(* IEC 61131-3 sources: volt/packages/volt-lsp-iec/test-corpus/pro2193/Device/Plc Logic/Application/09 Misc/Library Manager/SysTask, 36 files *)

(* ---- PFSYS_TASK_EXCEPTIONHANDLER.dut ---- *)
TYPE PFSYS_TASK_EXCEPTIONHANDLER : POINTER TO BYTE;
END_TYPE

(* ---- PFSYS_TASK_FUNCTION.dut ---- *)
TYPE PFSYS_TASK_FUNCTION : POINTER TO BYTE;
END_TYPE

(* ---- REGCONTEXT.dut ---- *)
TYPE REGCONTEXT :
STRUCT
	ULIP : __UXINT;
	ULBP : __UXINT;
	ULSP : __UXINT;
END_STRUCT
END_TYPE

(* ---- SYS_TASK_INFO.dut ---- *)
TYPE SYS_TASK_INFO :
STRUCT
	UIOSHANDLE : RTS_IEC_HANDLE;
	ISTATE : DINT;
	IOLDSTATE : DINT;
	TP : SYS_TASK_PARAM;
	ULCYCLETIME : UDINT;
	ULCYCLESTART : UDINT;
	ULPRIORITY : UDINT;
	ULOSPRIORITY : UDINT;
	ULINTERVAL : UDINT;
	ULSTACKSIZE : UDINT;
	PFUNCTION : PFSYS_TASK_FUNCTION;
	SZNAME : STRING(SYSTASK_MAX_NAME_LEN);
	PEXCEPTIONHANDLER : PFSYS_TASK_EXCEPTIONHANDLER;
	CONTEXT : RegContext;
	PCPPINSTANCE : POINTER TO BYTE;
	POSSPECIFIC : POINTER TO BYTE;
	ULFEATURE : DWORD;
END_STRUCT
END_TYPE

(* ---- SYS_TASK_PARAM.dut ---- *)
TYPE SYS_TASK_PARAM :
STRUCT
	HTASK : RTS_IEC_HANDLE;
	BEXIT : DINT;
	ULINTERVAL : UDINT;
	PPARAM : POINTER TO BYTE;
END_STRUCT
END_TYPE

(* ---- FEATUREFLAGS.gvl ---- *)
VAR_GLOBAL
	SYSTASK_FF_NONE : DWORD := 16#0;
	SYSTASK_FF_AUTORELEASEONEXIT : DWORD := 16#1;
END_VAR

(* ---- GVL.gvl ---- *)
VAR_GLOBAL
	SYSTASK_MAX_NAME_LEN : UDINT := 19;
END_VAR

(* ---- TASKPRIORITIES.gvl ---- *)
VAR_GLOBAL
	TASKPRIO_RANGE : UDINT := 255;
	TASKPRIO_SEGMENT : UDINT := 32;
	TASKPRIO_MAX : UDINT := 0;
	TASKPRIO_SYSTEM_BASE : UDINT := 0;
	TASKPRIO_SYSTEM_END : UDINT := 31;
	TASKPRIO_REALTIME_BASE : UDINT := 32;
	TASKPRIO_REALTIME_END : UDINT := 63;
	TASKPRIO_HIGH_BASE : UDINT := 64;
	TASKPRIO_HIGH_END : UDINT := 95;
	TASKPRIO_ABOVENORMAL_BASE : UDINT := 96;
	TASKPRIO_ABOVENORMAL_END : UDINT := 127;
	TASKPRIO_NORMAL_BASE : UDINT := 128;
	TASKPRIO_NORMAL_END : UDINT := 159;
	TASKPRIO_BELOWNORMAL_BASE : UDINT := 160;
	TASKPRIO_BELOWNORMAL_END : UDINT := 191;
	TASKPRIO_LOW_BASE : UDINT := 192;
	TASKPRIO_LOW_END : UDINT := 223;
	TASKPRIO_LOWEST_BASE : UDINT := 224;
	TASKPRIO_LOWEST_END : UDINT := 255;
	TASKPRIO_IDLE : UDINT := 255;
	TASKPRIO_MIN : UDINT := 255;
END_VAR

(* ---- SYSTASKAUTORELEASEONEXIT.pou ---- *)
FUNCTION SYSTASKAUTORELEASEONEXIT : RTS_IEC_RESULT
VAR_INPUT
	HTASK : RTS_IEC_HANDLE;
END_VAR
END_FUNCTION

(* ---- SYSTASKCHECKSTACK.pou ---- *)
FUNCTION SYSTASKCHECKSTACK : RTS_IEC_RESULT
VAR_INPUT
	HTASK : RTS_IEC_HANDLE;
	PULMAXDEPTH : POINTER TO UDINT;
END_VAR
END_FUNCTION

(* ---- SYSTASKCREATE.pou ---- *)
FUNCTION SYSTASKCREATE : RTS_IEC_RESULT
VAR_INPUT
	PSZTASKNAME : REFERENCE TO STRING;
	PFUNCTION : PFSYS_TASK_FUNCTION;
	PPARAM : POINTER TO SYS_TASK_PARAM;
	ULPRIORITY : UDINT;
	ULINTERVAL : UDINT;
	ULSTACKSIZE : UDINT;
	PEXCEPTIONHANDLER : PFSYS_TASK_EXCEPTIONHANDLER;
	PHTASKHANDLE : POINTER TO RTS_IEC_HANDLE;
END_VAR
END_FUNCTION

(* ---- SYSTASKCREATE2.pou ---- *)
FUNCTION SYSTASKCREATE2 : RTS_IEC_HANDLE
VAR_INPUT
	PSZTASKNAME : REFERENCE TO STRING;
	PFUNCTION : PFSYS_TASK_FUNCTION;
	PPARAM : POINTER TO SYS_TASK_PARAM;
	ULPRIORITY : UDINT;
	ULINTERVAL : UDINT;
	ULSTACKSIZE : UDINT;
	PEXCEPTIONHANDLER : PFSYS_TASK_EXCEPTIONHANDLER;
	PRESULT : POINTER TO RTS_IEC_RESULT;
END_VAR
END_FUNCTION

(* ---- SYSTASKDESTROY.pou ---- *)
FUNCTION SYSTASKDESTROY : RTS_IEC_RESULT
VAR_INPUT
	HTASK : RTS_IEC_HANDLE;
END_VAR
END_FUNCTION

(* ---- SYSTASKEND.pou ---- *)
FUNCTION SYSTASKEND : RTS_IEC_RESULT
VAR_INPUT
	HTASK : RTS_IEC_HANDLE;
	ULEXITCODE : UDINT;
END_VAR
END_FUNCTION

(* ---- SYSTASKENTER.pou ---- *)
FUNCTION SYSTASKENTER : RTS_IEC_RESULT
VAR_INPUT
	HTASK : RTS_IEC_HANDLE;
END_VAR
END_FUNCTION

(* ---- SYSTASKEXIT.pou ---- *)
FUNCTION SYSTASKEXIT : RTS_IEC_RESULT
VAR_INPUT
	HTASK : RTS_IEC_HANDLE;
	ULTIMEOUTMS : UDINT;
END_VAR
END_FUNCTION

(* ---- SYSTASKGENERATEEXCEPTION.pou ---- *)
FUNCTION SYSTASKGENERATEEXCEPTION : RTS_IEC_RESULT
VAR_INPUT
	ULTASKOSHANDLE : RTS_IEC_HANDLE;
	ULEXCEPTION : UDINT;
	CONTEXT : RegContext;
END_VAR
END_FUNCTION

(* ---- SYSTASKGETCONTEXT.pou ---- *)
FUNCTION SYSTASKGETCONTEXT : RTS_IEC_RESULT
VAR_INPUT
	HTASK : RTS_IEC_HANDLE;
	PCONTEXT : POINTER TO RegContext;
END_VAR
END_FUNCTION

(* ---- SYSTASKGETCURRENT.pou ---- *)
FUNCTION SYSTASKGETCURRENT : RTS_IEC_RESULT
VAR_INPUT
	PHTASK : POINTER TO RTS_IEC_HANDLE;
END_VAR
END_FUNCTION

(* ---- SYSTASKGETCURRENTOSHANDLE.pou ---- *)
FUNCTION SYSTASKGETCURRENTOSHANDLE : RTS_IEC_RESULT
VAR_INPUT
	PUITASKOSHANDLE : POINTER TO RTS_IEC_HANDLE;
END_VAR
END_FUNCTION

(* ---- SYSTASKGETINFO.pou ---- *)
FUNCTION SYSTASKGETINFO : RTS_IEC_RESULT
VAR_INPUT
	HTASK : RTS_IEC_HANDLE;
	PPINFO : POINTER TO POINTER TO SYS_TASK_INFO;
END_VAR
END_FUNCTION

(* ---- SYSTASKGETINTERVAL.pou ---- *)
FUNCTION SYSTASKGETINTERVAL : RTS_IEC_RESULT
VAR_INPUT
	HTASK : RTS_IEC_HANDLE;
END_VAR
VAR_IN_OUT
	PULINTERVAL : UDINT;
END_VAR
END_FUNCTION

(* ---- SYSTASKGETNAME.pou ---- *)
FUNCTION SYSTASKGETNAME : POINTER TO STRING
VAR_INPUT
	HTASK : RTS_IEC_HANDLE;
	PRESULT : POINTER TO RTS_IEC_RESULT;
END_VAR
END_FUNCTION

(* ---- SYSTASKGETOSHANDLE.pou ---- *)
FUNCTION SYSTASKGETOSHANDLE : RTS_IEC_HANDLE
VAR_INPUT
	HTASK : RTS_IEC_HANDLE;
END_VAR
END_FUNCTION

(* ---- SYSTASKGETOSPRIORITY.pou ---- *)
FUNCTION SYSTASKGETOSPRIORITY : RTS_IEC_RESULT
VAR_INPUT
	HTASK : RTS_IEC_HANDLE;
	PULOSPRIORITY : POINTER TO UDINT;
END_VAR
END_FUNCTION

(* ---- SYSTASKGETPRIORITY.pou ---- *)
FUNCTION SYSTASKGETPRIORITY : RTS_IEC_RESULT
VAR_INPUT
	HTASK : RTS_IEC_HANDLE;
	PULPRIORITY : POINTER TO UDINT;
END_VAR
END_FUNCTION

(* ---- SYSTASKJOIN.pou ---- *)
FUNCTION SYSTASKJOIN : RTS_IEC_RESULT
VAR_INPUT
	HTASKTOJOIN : RTS_IEC_HANDLE;
	ULTIMEOUTMS : UDINT;
END_VAR
END_FUNCTION

(* ---- SYSTASKLEAVE.pou ---- *)
FUNCTION SYSTASKLEAVE : RTS_IEC_RESULT
VAR_INPUT
	HTASK : RTS_IEC_HANDLE;
END_VAR
END_FUNCTION

(* ---- SYSTASKRESUME.pou ---- *)
FUNCTION SYSTASKRESUME : RTS_IEC_RESULT
VAR_INPUT
	HTASK : RTS_IEC_HANDLE;
END_VAR
END_FUNCTION

(* ---- SYSTASKSETEXIT.pou ---- *)
FUNCTION SYSTASKSETEXIT : RTS_IEC_RESULT
VAR_INPUT
	HTASK : RTS_IEC_HANDLE;
END_VAR
END_FUNCTION

(* ---- SYSTASKSETINTERVAL.pou ---- *)
FUNCTION SYSTASKSETINTERVAL : RTS_IEC_RESULT
VAR_INPUT
	HTASK : RTS_IEC_HANDLE;
	ULINTERVAL : UDINT;
END_VAR
END_FUNCTION

(* ---- SYSTASKSETPRIORITY.pou ---- *)
FUNCTION SYSTASKSETPRIORITY : RTS_IEC_RESULT
VAR_INPUT
	HTASK : RTS_IEC_HANDLE;
	ULPRIORITY : UDINT;
END_VAR
END_FUNCTION

(* ---- SYSTASKSUSPEND.pou ---- *)
FUNCTION SYSTASKSUSPEND : RTS_IEC_RESULT
VAR_INPUT
	HTASK : RTS_IEC_HANDLE;
END_VAR
END_FUNCTION

(* ---- SYSTASKWAITINTERVAL.pou ---- *)
FUNCTION SYSTASKWAITINTERVAL : RTS_IEC_RESULT
VAR_INPUT
	HTASK : RTS_IEC_HANDLE;
END_VAR
END_FUNCTION

(* ---- SYSTASKWAITSLEEP.pou ---- *)
FUNCTION SYSTASKWAITSLEEP : RTS_IEC_RESULT
VAR_INPUT
	HTASK : RTS_IEC_HANDLE;
	ULMILLISECONDS : UDINT;
END_VAR
END_FUNCTION

(* ---- SYSTASKWAITSLEEPUS.pou ---- *)
FUNCTION SYSTASKWAITSLEEPUS : RTS_IEC_RESULT
VAR_INPUT
	HTASK : RTS_IEC_HANDLE;
END_VAR
VAR_IN_OUT
	PTSLEEPUS : SYSTIME;
END_VAR
END_FUNCTION
